// TIA Portal V15.1 export
// export: Created 2024-05-17T05:38:25.0999793Z, ExportSetting WithDefaults, DisplayName Totally Integrated Automation Portal, DisplayVersion V15.1 Update 5, DisplayName TIA Portal Openness, DisplayVersion V15.1 Update 5, DisplayName SINAMICS Startdrive Advanced, DisplayVersion V15.1, DisplayName G130, G150, S120, S150, SINAMICS MV, S210, DisplayVersion V15.1, DisplayName G110M, G120, G120C, G120D, G120P, DisplayVersion V15.1, DisplayName STEP 7 Professional, DisplayVersion V15.1 Update 5, DisplayName STEP 7 Safety, DisplayVersion V15.1, DisplayName WinCC Professional, DisplayVersion V15.1 Update 5, DisplayName SIMATIC Visualization Architect, DisplayVersion V15.1
FUNCTION_BLOCK "LPartSensor"   // FB1614, FBD
TITLE = LPartDet
{ S7_Optimized_Access := 'FALSE' }
AUTHOR : VCC
FAMILY : ToolEqp
NAME : LPartSen
VERSION : 1.0
// ===============================================================================
// This module handles a partdetection with all his functions and alarms
// Functions are DetCheckOn, DetCheckOff and EnableAlarm
// Outputs are DetAlarm and DetOn signal
// ===============================================================================
// stored: AutoNumber false, IsIECCheckEnabled false, SetENOAutomatically False, UDAEnableTagReadback false
   VAR_INPUT
      I_SignalCheckOn { ExternalAccessible := 'False'; ExternalVisible := 'False'; ExternalWritable := 'False'} : Bool;   // Signal to check signal is on
      I_Signal { ExternalAccessible := 'False'; ExternalVisible := 'False'; ExternalWritable := 'False'} : Bool;   // Actual input from sensor
      I_SignalCheckOff { ExternalAccessible := 'False'; ExternalVisible := 'False'; ExternalWritable := 'False'} : Bool;   // Signal to check signal is off
      I_Simulate : Bool;   // Simulation mode
      I_AlarmClass { ExternalAccessible := 'False'; ExternalVisible := 'False'; ExternalWritable := 'False'} : Char;   // Alarm class -> A - B - C - D or E
      I_EnableAlarm { ExternalAccessible := 'False'; ExternalVisible := 'False'; ExternalWritable := 'False'} : Bool;   // Enable alarms
      I_AlarmResetPB { ExternalAccessible := 'False'; ExternalVisible := 'False'; ExternalWritable := 'False'} : Bool;   // Alarm reset pushbutton is activated
   END_VAR
   VAR_OUTPUT
      O_DetOn { ExternalAccessible := 'False'; ExternalVisible := 'False'; ExternalWritable := 'False'} : Bool;   // Detection signal to use in program
      O_DetAlmReqOn { ExternalAccessible := 'False'; ExternalVisible := 'False'; ExternalWritable := 'False'} : Bool;   // Request on alarm
      O_DetAlmReqOff { ExternalAccessible := 'False'; ExternalVisible := 'False'; ExternalWritable := 'False'} : Bool;   // Request off alarm
      O_DetSumAlm { ExternalAccessible := 'False'; ExternalVisible := 'False'; ExternalWritable := 'False'} : Bool;   // Request on or request off signal active
      O_AlarmABCondition { ExternalAccessible := 'False'; ExternalVisible := 'False'; ExternalWritable := 'False'} : Bool;   // Alarm AB condition
      H_IAnim { ExternalAccessible := 'False'; ExternalVisible := 'False'; ExternalWritable := 'False'} : Word;   // For animation of the icon
   END_VAR
   VAR DB_SPECIFIC
      H_Out : Struct   // HMI
         Anim : Word;   // HMI Animation of the object
         DBnr : Int;   // HMI Animation DB number
      END_STRUCT;
      DetCheckOnAlarm { ExternalAccessible := 'False'; ExternalVisible := 'False'; ExternalWritable := 'False'} : Bool;   // Detection is not on
      DetCheckOffAlarm { ExternalAccessible := 'False'; ExternalVisible := 'False'; ExternalWritable := 'False'} : Bool;   // Detection is not off
      DetOn { ExternalAccessible := 'False'; ExternalVisible := 'False'; ExternalWritable := 'False'} : Bool;   // Detection on
      DetAlarm { ExternalAccessible := 'False'; ExternalVisible := 'False'; ExternalWritable := 'False'} : Bool;   // Detection alarm
      AlarmCondReqOn { ExternalAccessible := 'False'; ExternalVisible := 'False'; ExternalWritable := 'False'} : Bool;   // Alarm condition
      AlarmCondReqOff { ExternalAccessible := 'False'; ExternalVisible := 'False'; ExternalWritable := 'False'} : Bool;   // Alarm condition
      AlarmClass_A { ExternalAccessible := 'False'; ExternalVisible := 'False'; ExternalWritable := 'False'} : Bool;   // The alarm is from alarm class A
      AlarmClass_B { ExternalAccessible := 'False'; ExternalVisible := 'False'; ExternalWritable := 'False'} : Bool;   // The alarm is from alarm class B
      AlarmClass_C { ExternalAccessible := 'False'; ExternalVisible := 'False'; ExternalWritable := 'False'} : Bool;   // The alarm is from alarm class C
      AlarmClass_D { ExternalAccessible := 'False'; ExternalVisible := 'False'; ExternalWritable := 'False'} : Bool;   // The alarm is from alarm class D
      AlarmClass_E { ExternalAccessible := 'False'; ExternalVisible := 'False'; ExternalWritable := 'False'} : Bool;   // The alarm is from alarm class E
      DBnr { ExternalAccessible := 'False'; ExternalVisible := 'False'; ExternalWritable := 'False'} : Int;   // HMI DB number
   END_VAR
BEGIN

NETWORK
TITLE = **** 1 - Inputs **** DB number
// DB number
      L     DINO;
      T     #DBnr;

NETWORK
TITLE = **** 1 - Inputs **** Alarm class
// Alarm class
// Alarm class = E
      L     #I_AlarmClass;
      L     'E';
      ==I;
      =     #AlarmClass_E;

// Alarm class = D
      L     #I_AlarmClass;
      L     'D';
      ==I;
      =     #AlarmClass_D;

// Alarm class = C
      L     #I_AlarmClass;
      L     'C';
      ==I;
      =     #AlarmClass_C;

// Alarm class = B
      L     #I_AlarmClass;
      L     'B';
      ==I;
      =     #AlarmClass_B;

// Alarm class = A
      AN    #AlarmClass_B;
      AN    #AlarmClass_C;
      AN    #AlarmClass_D;
      AN    #AlarmClass_E;
      =     #AlarmClass_A;


REGION Network 3: **** 2.2 - Alarms - Alarm generation **** Condition alarm for active detection
   // Condition alarm for active detection
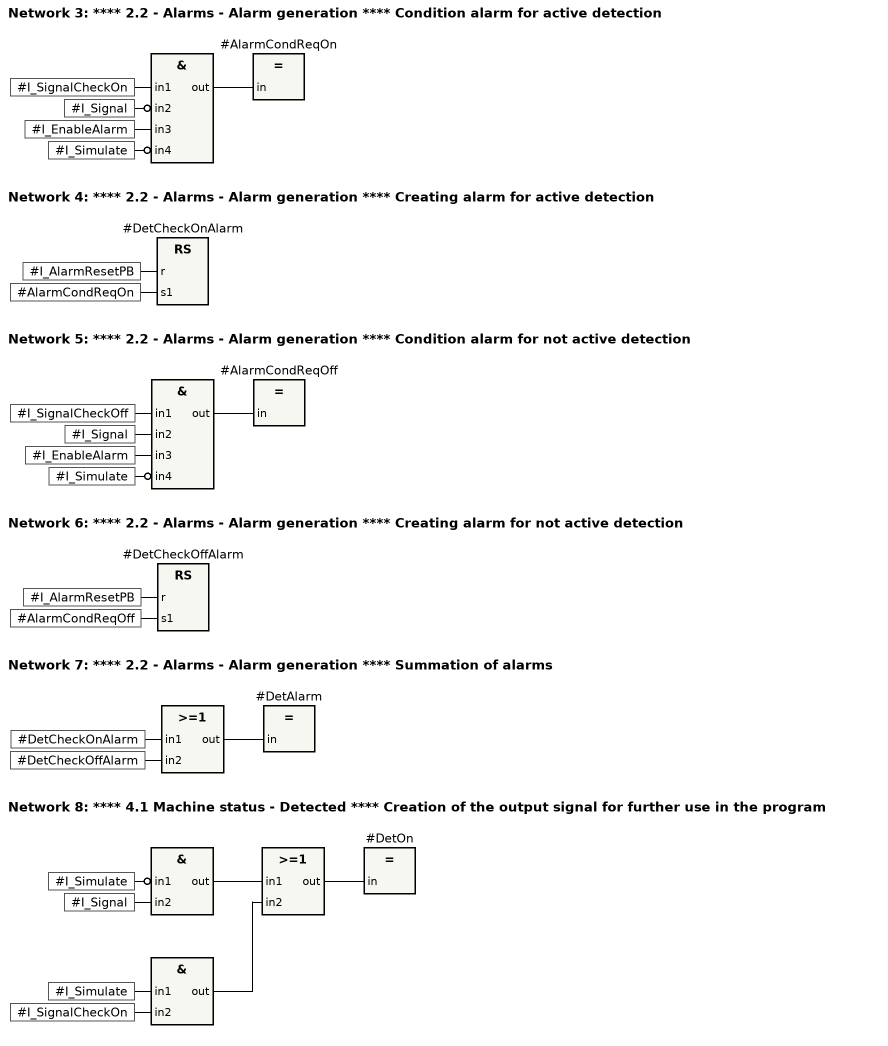
   #AlarmCondReqOn := #I_SignalCheckOn AND NOT #I_Signal AND #I_EnableAlarm AND NOT #I_Simulate;
END_REGION

REGION Network 4: **** 2.2 - Alarms - Alarm generation **** Creating alarm for active detection
   // Creating alarm for active detection
   IF #I_AlarmResetPB THEN
       #DetCheckOnAlarm := FALSE;   // RS flip-flop
   END_IF;
   IF #AlarmCondReqOn THEN #DetCheckOnAlarm := TRUE; END_IF;
END_REGION

REGION Network 5: **** 2.2 - Alarms - Alarm generation **** Condition alarm for not active detection
   // Condition alarm for not active detection
   #AlarmCondReqOff := #I_SignalCheckOff AND #I_Signal AND #I_EnableAlarm AND NOT #I_Simulate;
END_REGION

REGION Network 6: **** 2.2 - Alarms - Alarm generation **** Creating alarm for not active detection
   // Creating alarm for not active detection
   IF #I_AlarmResetPB THEN
       #DetCheckOffAlarm := FALSE;   // RS flip-flop
   END_IF;
   IF #AlarmCondReqOff THEN #DetCheckOffAlarm := TRUE; END_IF;
END_REGION

REGION Network 7: **** 2.2 - Alarms - Alarm generation **** Summation of alarms
   // Summation of alarms
   #DetAlarm := #DetCheckOnAlarm OR #DetCheckOffAlarm;
END_REGION

REGION Network 8: **** 4.1 Machine status - Detected **** Creation of the output signal for further use in the program
   // Creation of the output signal for further use in the program
   #DetOn := (NOT #I_Simulate AND #I_Signal) OR (#I_Simulate AND #I_SignalCheckOn);
END_REGION

REGION Network 9: **** 4.6 - Machine Status - Indications **** Icon animation
   // Icon animation
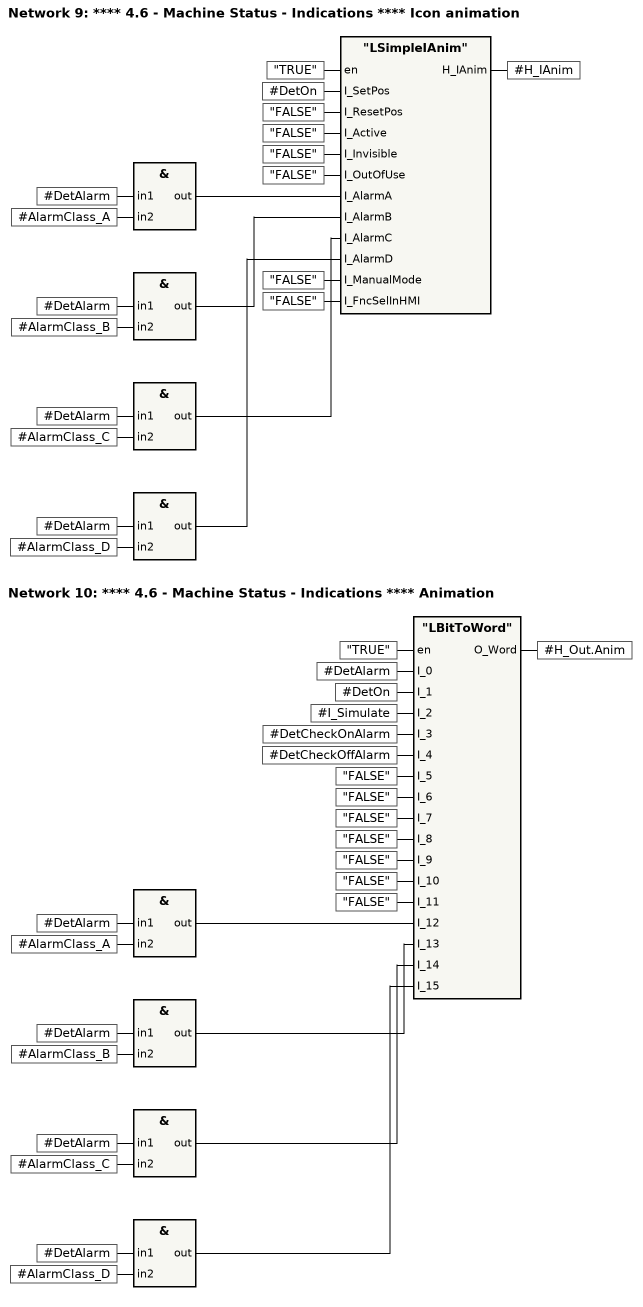
   IF "TRUE" THEN
       "LSimpleIAnim"(I_SetPos := #DetOn,
                      I_ResetPos := "FALSE",
                      I_Active := "FALSE",
                      I_Invisible := "FALSE",
                      I_OutOfUse := "FALSE",
                      I_AlarmA := #DetAlarm AND #AlarmClass_A,
                      I_AlarmB := #DetAlarm AND #AlarmClass_B,
                      I_AlarmC := #DetAlarm AND #AlarmClass_C,
                      I_AlarmD := #DetAlarm AND #AlarmClass_D,
                      I_ManualMode := "FALSE",
                      I_FncSelInHMI := "FALSE",
                      H_IAnim => #H_IAnim);
   END_IF;
END_REGION

REGION Network 10: **** 4.6 - Machine Status - Indications **** Animation
   // Animation
   IF "TRUE" THEN
       "LBitToWord"(I_0 := #DetAlarm,
                    I_1 := #DetOn,
                    I_2 := #I_Simulate,
                    I_3 := #DetCheckOnAlarm,
                    I_4 := #DetCheckOffAlarm,
                    I_5 := "FALSE",
                    I_6 := "FALSE",
                    I_7 := "FALSE",
                    I_8 := "FALSE",
                    I_9 := "FALSE",
                    I_10 := "FALSE",
                    I_11 := "FALSE",
                    I_12 := #DetAlarm AND #AlarmClass_A,
                    I_13 := #DetAlarm AND #AlarmClass_B,
                    I_14 := #DetAlarm AND #AlarmClass_C,
                    I_15 := #DetAlarm AND #AlarmClass_D,
                    O_Word => #H_Out.Anim);
   END_IF;
END_REGION

REGION Network 11: **** 4.6 - Machine status - Indications **** Animation DB number
   // Animation DB number
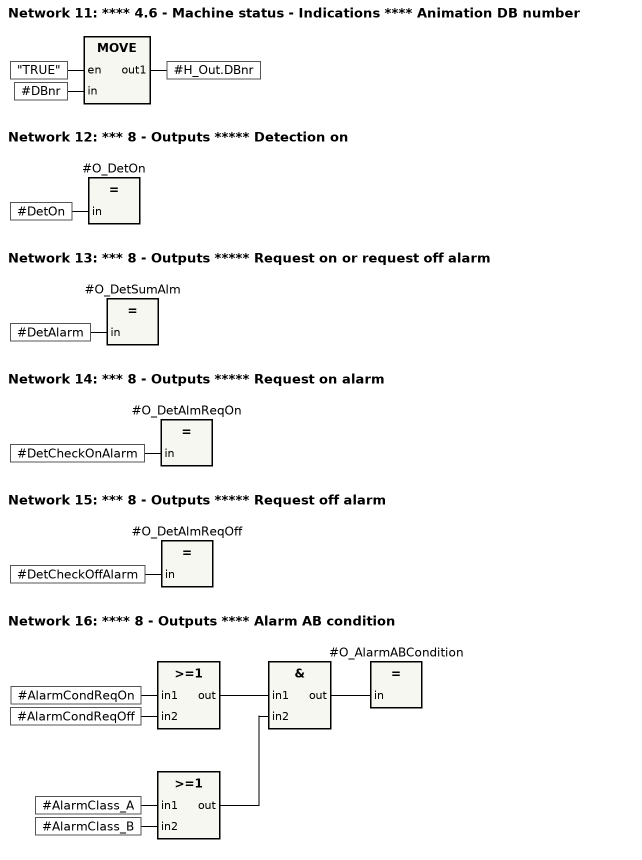
   IF "TRUE" THEN #H_Out.DBnr := #DBnr; END_IF;
END_REGION

REGION Network 12: *** 8 - Outputs ***** Detection on
   // Detection on
   #O_DetOn := #DetOn;
END_REGION

REGION Network 13: *** 8 - Outputs ***** Request on or request off alarm
   // Request on or request off alarm
   #O_DetSumAlm := #DetAlarm;
END_REGION

REGION Network 14: *** 8 - Outputs ***** Request on alarm
   // Request on alarm
   #O_DetAlmReqOn := #DetCheckOnAlarm;
END_REGION

REGION Network 15: *** 8 - Outputs ***** Request off alarm
   // Request off alarm
   #O_DetAlmReqOff := #DetCheckOffAlarm;
END_REGION

REGION Network 16: **** 8 - Outputs **** Alarm AB condition
   // Alarm AB condition
   #O_AlarmABCondition := (#AlarmCondReqOn OR #AlarmCondReqOff) AND (#AlarmClass_A OR #AlarmClass_B);
END_REGION
END_FUNCTION_BLOCK
